Fanuc KAREL source: kt00044.KL

-- PROVISIONAL review KL for V770-1; original PC SHA256 11ae911f201d9c9bd539b844d98a7e79d24acca0a1f4340bfb8e0b654d12700f
-- Incomplete behavior may be omitted. Consult companion uncertainty JSON. Do not deploy.
PROGRAM KT00044
%NOLOCKGROUP
VAR
  R1 : REAL
  R2 : REAL
  OUT : REAL
BEGIN
  -- UNRESOLVED_PC offsets 5-16; opcodes 2E,23
  -- UNRESOLVED_PC offsets 21-32; opcodes 2E,23
  -- UNRESOLVED_PC offsets 37-48; opcodes 2E,23
  -- UNRESOLVED_PC offsets 53-64; opcodes 2E,23
  -- UNRESOLVED_PC offsets 69-88; opcodes 21,21,6A,23
  -- UNRESOLVED_PC offsets 93-97; opcodes 7F
END KT00044
